// Mitsubishi GX Works2 project: 펑션라벨으요   PLC: Q02/Q02H

PROGRAM MAIN
VAR
  자기_1 : 자기;
  자기_2 : 자기;
  인터록_1 : 인터록;
  업카운트_1 : 업카운트;
  다운카운트_1 : 다운카운트;
  응용_1 : 응용;
END_VAR
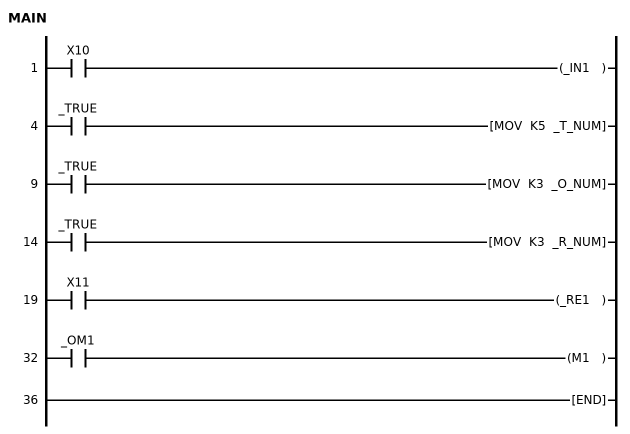
; FB BLK START 응용(응용_1)
1     LD      X10
      OUT     _IN1
4     LD      _TRUE
      MOV     K5 _T_NUM
9     LD      _TRUE
      MOV     K3 _O_NUM
14    LD      _TRUE
      MOV     K3 _R_NUM
19    LD      X11
      OUT     _RE1
; FB START
; FB_NAME 응용
; INSTANCE_NAME 응용_1
; FB IN_B:IN1
; FB OUT_OM1:B
; FB IN_W:T_NUM
; FB IN_W:O_NUM
; FB IN_W:R_NUM
; FB IN_B:RE1
; FB END
32    LD      _OM1
      OUT     M1
; FB BLK END
36    END
END_PROGRAM

FUNCTION_BLOCK 자기
VAR_INPUT
  INN1 : BOOL;
  INN2 : BOOL;
END_VAR
VAR_OUTPUT
  OUTT : BOOL;
END_VAR
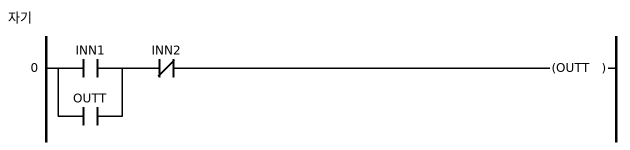
0     LD      INN1
      OR      OUTT
      ANI     INN2
      OUT     OUTT
END_FUNCTION_BLOCK

FUNCTION_BLOCK 인터록
VAR_INPUT
  ITIN1 : BOOL;
  ITIN2 : BOOL;
  ITIN3 : BOOL;
END_VAR
VAR_OUTPUT
  ITOUT1 : BOOL;
  ITOUT2 : BOOL;
END_VAR
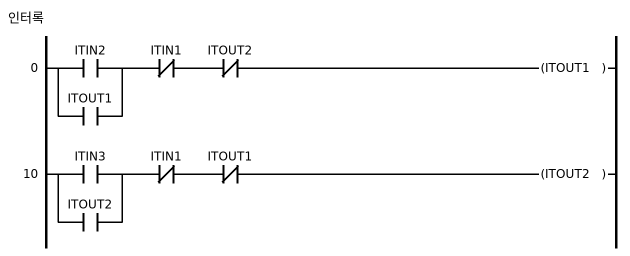
0     LD      ITIN2
      OR      ITOUT1
      ANI     ITIN1
      ANI     ITOUT2
      OUT     ITOUT1
10    LD      ITIN3
      OR      ITOUT2
      ANI     ITIN1
      ANI     ITOUT1
      OUT     ITOUT2
END_FUNCTION_BLOCK

FUNCTION_BLOCK 업카운트
VAR_INPUT
  CIN : BOOL;
  Re : BOOL;
END_VAR
VAR_OUTPUT
  COUT : BOOL;
END_VAR
VAR_INPUT
  PV : INT;
END_VAR
VAR_OUTPUT
  CV : INT;
END_VAR
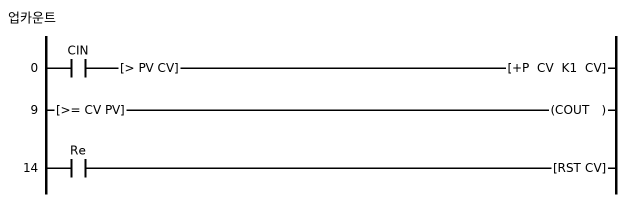
0     LD      CIN
      AND>    PV CV
      +P      CV K1 CV
9     LD>=    CV PV
      OUT     COUT
14    LD      Re
      RST     CV
END_FUNCTION_BLOCK

FUNCTION_BLOCK 다운카운트
VAR_INPUT
  C_in : BOOL;
  C_num : INT;
  C_re : BOOL;
END_VAR
VAR_OUTPUT
  C_out : BOOL;
  C_mem : INT;
END_VAR
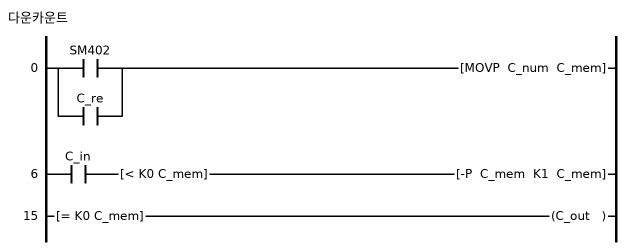
0     LD      SM402
      OR      C_re
      MOVP    C_num C_mem
6     LD      C_in
      AND<    K0 C_mem
      -P      C_mem K1 C_mem
15    LD=     K0 C_mem
      OUT     C_out
END_FUNCTION_BLOCK

FUNCTION_BLOCK 응용
VAR_INPUT
  IN1 : BOOL;
  T_NUM : INT;
  O_NUM : INT;
  R_NUM : INT;
  RE1 : BOOL;
END_VAR
VAR_OUTPUT
  OM1 : BOOL;
END_VAR
VAR
  WT1 : TIMER;
  WT2 : TIMER;
  CC1 : COUNTER;
END_VAR
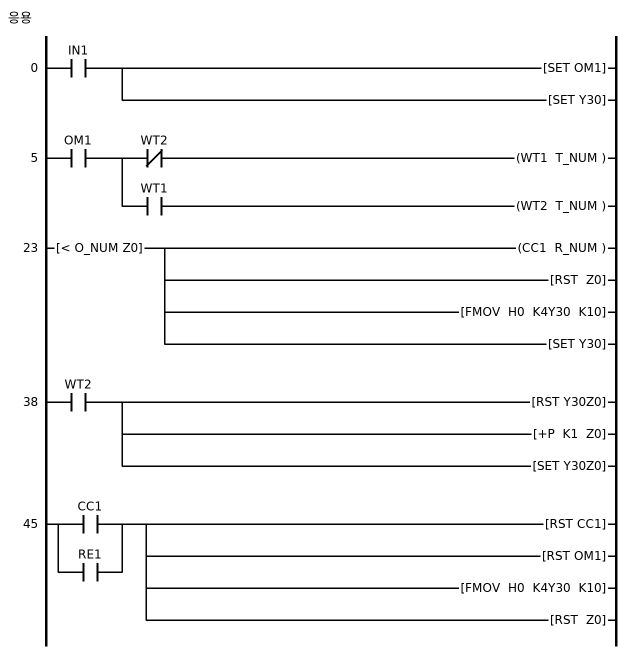
0     LD      IN1
      SET     OM1
      SET     Y30
5     LD      OM1
      MPS
      ANI     WT2
      OUT     WT1 T_NUM
      MPP
      AND     WT1
      OUT     WT2 T_NUM
23    LD<     O_NUM Z0
      OUT     CC1 R_NUM
      RST     Z0
      FMOV    H0 K4Y30 K10
      SET     Y30
38    LD      WT2
      RST     Y30Z0
      +P      K1 Z0
      SET     Y30Z0
45    LD      CC1
      OR      RE1
      RST     CC1
      RST     OM1
      FMOV    H0 K4Y30 K10
      RST     Z0
END_FUNCTION_BLOCK
